(*
	Y:2016	M:05	D:20
	T:INTERFACE		N:GENERIC COMMUNICATION INTERFACE
*)
INTERFACE IFC_GENERIC_COMMUNICATION_INTERFACE

METHOD Close_Connection : RETURN_CODE
VAR_INPUT
END_VAR
END_METHOD

METHOD Open_Connection : RETURN_CODE
VAR_INPUT
END_VAR
END_METHOD

METHOD Read : RETURN_CODE
VAR_INPUT
	Configuration : S_GCI_CONFIG;
END_VAR
END_METHOD

METHOD Write : RETURN_CODE
VAR_INPUT
	Configuration : S_GCI_CONFIG;
END_VAR
END_METHOD

END_INTERFACE

(* stored: Version 1.1.0.1, ProductVersion 3.1.4019.2
   Itf IFC_GENERIC_COMMUNICATION_INTERFACE: Id {025bd610-72e5-47fb-8e6c-9d00611370f5}
   Method Close_Connection: Id {f2af6587-9985-4073-a448-95fd488a7b24}
   Method Open_Connection: Id {bd81e16c-fef7-4eee-ac3c-d5841221af71}
   Method Read: Id {19c79a54-9157-436c-801e-b935e8fe99d5}
   Method Write: Id {548b3c14-dc8d-4a49-ae41-d0957254011e} *)
